// TwinCAT 3 PLC project Library
// Title: LCLS Sample Delivery
// Company: SLAC - LCLS
// ProjectVersion: 0.0.0
// ProgramVersion: 3.1.4023.0
// libraries:
//   LCLS Vacuum, * (SLAC - LCLS)
//   PMPS, * (SLAC - LCLS)
//   Tc2_EtherCAT, * (Beckhoff Automation GmbH)
//   Tc2_MC2, * (Beckhoff Automation GmbH)
//   Tc2_ModbusSrv, * (Beckhoff Automation GmbH)
//   Tc2_SerialCom, * (Beckhoff Automation GmbH)
//   Tc2_Standard, * (Beckhoff Automation GmbH)
//   Tc2_SUPS, * (Beckhoff Automation GmbH)
//   Tc2_System, * (Beckhoff Automation GmbH)
//   Tc2_Utilities, * (Beckhoff Automation GmbH)
//   Tc3_Module, * (Beckhoff Automation GmbH)
//   TcUnit, * (www.tcunit.org)
//   LCLS General,2.12.0,SLAC
// project tree:
//   DUTs/ALI/ E_AxisMoveMode.TcDUT (not stored), E_CTRL_MODE.TcDUT (not stored), E_PropValveFBState.TcDUT (not stored), HMI_PropValveCtrlState.TcDUT (not stored), ST_ALI.TcDUT (not stored), ST_ManipAxis.TcDUT (not stored), ST_PIDParams.TcDUT (not stored), ST_PressureController.TcDUT (not stored), ST_PropValveMKS253.TcDUT (not stored)
//   DUTs/Bronkhorst/ E_BHElFlowUnit.TcDUT (not stored), ST_BhElFlow.TcDUT (not stored)
//   DUTs/ E_AxisMotionState.TcDUT (not stored), ST_ManifoldValve.TcDUT (not stored), ST_Proportionair.TcDUT (not stored), ST_RegDeadbandControls.TcDUT (not stored), ST_Regulator.TcDUT (not stored), ST_SelectorM3.TcDUT (not stored), ST_Shaker.TcDUT (not stored), ST_ShakerControls.TcDUT (not stored), ST_Strings.TcDUT (not stored)
//   DUTs/General/ E_CTRL_MODE_1.TcDUT (not stored)
//   DUTs/IO_Structs/ ST_ALIIO.TcDUT (not stored), ST_M3DeviceBaseIO.TcDUT (not stored), ST_SerialComm.TcDUT (not stored)
//   DUTs/RCC/ E_RCC_PUMP_SM_STATES.TcDUT, E_RCC_STATES.TcDUT (not stored), ST_RCC.TcDUT
//   DUTs/Sensirion/ E_SensirionFMMode.TcTLEO (not stored), ST_SensirionFM.TcDUT (not stored), ST_SensirionFMControl.TcDUT (not stored), ST_SensirionFMStatus.TcDUT (not stored)
//   DUTs/TEC/ ST_TECControl.TcDUT (not stored), ST_TECStatus.TcDUT (not stored)
//   DUTs/Vici/EPS/ E_VICI_PORT_EPS.TcDUT, E_VICI_EPS_PORT_STATUS.TcDUT
//   DUTs/Vici/ ST_12ViciValveSampleNames.TcDUT, ST_4PViciValveSampleNames.TcDUT, ST_ViciControl.TcDUT (not stored), ST_ViciStatus.TcDUT (not stored)
//   GVLs/ GVL_SAMPLE.TcGVL (not stored)
//   / PlcTask.TcTTO (not stored)
//   POUs/ALI/ FB_ALI.TcPOU (not stored), FB_ManipAxis.TcPOU (not stored), FB_PID_EXT.TcPOU (not stored), FB_PropValve.TcPOU (not stored), F_AxisRef_To_MSTA.TcPOU (not stored), MC_SmoothMover.TcPOU (not stored)
//   POUs/Bronkhorst/ FB_BronkhorstMFM.TcPOU (not stored)
//   POUs/DigitalOutput/ FB_SolenoidPair.TcPOU (not stored)
//   POUs/ EXAMPLE_DEPLOYMENT.TcPOU (not stored), PRG_TEST.TcPOU
//   POUs/GasManifold/ FB_GasManifold.TcPOU (not stored), FB_ManiValve.TcPOU (not stored)
//   POUs/Helpers/ FB_EcatDiag.TcPOU (not stored), FB_SelectorSync.TcPOU (not stored), FB_SerialCommWrapper.TcPOU (not stored), FB_ShiftByteArray.TcPOU (not stored)
//   POUs/PCM/ FB_MPV1.TcPOU, FB_PCM_AIO.TcPOU, FB_PressureControlModule.TcPOU (not stored)
//   POUs/RCC/ FB_RCC.TcPOU (not stored), FB_RCC_PUMP.TcPOU, FB_RCC_SM.TcPOU (not stored), FB_VRC_NC_OPNLS.TcPOU (not stored)
//   POUs/Regulators/ FB_ProportionairRegulator.TcPOU (not stored), FB_Regulator.TcPOU (not stored), F_rPressure.TcPOU (not stored)
//   POUs/Selectors/ FB_SelectorM3.TcPOU (not stored)
//   POUs/Sensirion/ FB_SenserionFlowMeter.TcPOU (not stored), FB_SensirionDriver.TcPOU (not stored), FB_SensirionTransaction.TcPOU (not stored), fSHDLCChecksum.TcPOU (not stored)
//   POUs/TEC/ FB_TECDriver.TcPOU (not stored), FB_TECTransaction.TcPOU (not stored)
//   POUs/Tests/ FB_RCC_TEST.TcPOU (not stored), FB_VICI_EPS_TEST.TcPOU
//   POUs/VICI/EPS/ FB_12PVICI_EPS.TcPOU, FB_4PVICI_EPS.TcPOU, FB_ViciValveEPS.TcPOU, FB_VICI_EPS_LOGIC.TcPOU
//   POUs/VICI/ FB_12PortVici.TcPOU, FB_4PortViciValve.TcPOU (not stored), FB_ViciDriver.TcPOU (not stored), FB_ViciTransaction.TcPOU (not stored), FB_ViciValve.TcPOU (not stored)
// real-time tasks:
//   TASK PlcTask: cycle T#10ms, priority 20, ADS port 350

// ---- DUTs/RCC/E_RCC_PUMP_SM_STATES.TcDUT
{attribute 'qualified_only'}
{attribute 'strict'}
TYPE E_RCC_PUMP_SM_STATES :
(
    IDLE := 0,
    PRESSURE := 1,
    VACUUM := 2,
    VENT := 3
);
END_TYPE

// ---- DUTs/RCC/ST_RCC.TcDUT
TYPE ST_RCC :
STRUCT
    {attribute 'pytmc' :='
        pv: Tinterval
        io: io
        autosave_pass0: VAL DESC
    '} // Time before cycle starts
    TInterval : REAL := 10;
    {attribute 'pytmc' :='
        pv: T1
        io: io
        autosave_pass0: VAL DESC
    '}
    T1 : REAL := 20;
    {attribute 'pytmc' :='
        pv: T2
        io: io
        autosave_pass0: VAL DESC
    '}
    T2 : REAL := 10;
    {attribute 'pytmc' :='
        pv: T3
        io: io
        autosave_pass0: VAL DESC
    '}
    T3 : REAL := 5;
    {attribute 'pytmc' :='
        pv: T4
        io: io
        autosave_pass0: VAL DESC
    '}
    T4 : REAL := 10;
    {attribute 'pytmc' :=' pv: RUNCLEAN'}
    bRunClean : BOOL := TRUE;

    {attribute 'pytmc' :=' pv: CLEAR_ERROR'}
    bClearError : BOOL := FALSE;
    {attribute 'pytmc' :=' pv: ERROR'}
    bError : BOOL := FALSE;
    {attribute 'pytmc' :=' pv: STOP_CYCLE'}
    bStop : BOOL := FALSE;

    {attribute 'pytmc' :=' pv: START_CYCLE'}
    bStartCycle : BOOL  := FALSE;

    {attribute 'pytmc' :='
        pv: ILK_Setpoint
        autosave_pass0: VAL DESC
     '}
    RCC_GCP_01_INTERLOCK_SETPOINT : REAL := 10;
    {attribute 'pytmc' :=' pv: OverrideMode '}
    xSystemOverrideMode_RCC : BOOL := FALSE;

    eCurrentState : INT := E_RCC_STATES.IDLE;

    {attribute 'pytmc' :='
        pv: RCC_RUNNING
        io: o
    '}
    bRunning : BOOL := FALSE;
    {attribute 'pytmc' :='
        pv: RCC_TIMER
        io: o
    '}
    tTimerReadBack : STRING := '';
    {attribute 'pytmc' :=' pv: sLogMessage '}
    sLogMessage : T_MaxString := '';

    RCC_VRC_01_OPEN_OK : BOOL;
    RCC_VRC_02_OPEN_OK : BOOL;
    RCC_VRC_03_OPEN_OK : BOOL;
    RCC_VRC_04_OPEN_OK : BOOL;

END_STRUCT
END_TYPE

// ---- DUTs/Vici/EPS/E_VICI_PORT_EPS.TcDUT
TYPE E_VICI_PORT_EPS :
STRUCT
    {attribute 'pytmc' := 'pv: stEPS'}
    stEPS : DUT_EPS;
    {attribute 'pytmc' := 'pv: ePortStatus'}
    ePortStatus : E_VICI_EPS_PORT_STATUS;
END_STRUCT
END_TYPE

// ---- DUTs/Vici/EPS/E_VICI_EPS_PORT_STATUS.TcDUT
{attribute 'qualified_only'}
{attribute 'strict'}
TYPE E_VICI_EPS_PORT_STATUS :
(
    ACTIVE := 0,
    UNLOCKED := 1,
    LOCKED := 2
);
END_TYPE

// ---- DUTs/Vici/ST_12ViciValveSampleNames.TcDUT
TYPE ST_12ViciValveSampleNames :
STRUCT
    {attribute 'pytmc' := '
        pv: 01
        io: io
        autosave_pass0: VAL DESC
     '}
     s1 : STRING;
     {attribute 'pytmc' := '
        pv: 02
        io: io
        autosave_pass0: VAL DESC
     '}
     s2 : STRING;
     {attribute 'pytmc' := '
        pv: 03
        io: io
        autosave_pass0: VAL DESC
     '}
     s3 : STRING;
     {attribute 'pytmc' := '
        pv: 04
        io: io
        autosave_pass0: VAL DESC
     '}
     s4 : STRING;
           {attribute 'pytmc' := '
        pv: 05
        io: io
        autosave_pass0: VAL DESC
     '}
     s5 : STRING;
     {attribute 'pytmc' := '
        pv: 06
        io: io
        autosave_pass0: VAL DESC
     '}
     s6 : STRING;
     {attribute 'pytmc' := '
        pv: 07
        io: io
        autosave_pass0: VAL DESC
     '}
     s7 : STRING;
     {attribute 'pytmc' := '
        pv: 08
        io: io
        autosave_pass0: VAL DESC
     '}
     s8 : STRING;
           {attribute 'pytmc' := '
        pv: 09
        io: io
        autosave_pass0: VAL DESC
     '}
     s9 : STRING;
     {attribute 'pytmc' := '
        pv: 10
        io: io
        autosave_pass0: VAL DESC
     '}
     s10 : STRING;
     {attribute 'pytmc' := '
        pv: 11
        io: io
        autosave_pass0: VAL DESC
     '}
     s11 : STRING;
     {attribute 'pytmc' := '
        pv: 12
        io: io
        autosave_pass0: VAL DESC
     '}
     s12 : STRING;
END_STRUCT
END_TYPE

// ---- DUTs/Vici/ST_4PViciValveSampleNames.TcDUT
TYPE ST_4PViciValveSampleNames :
STRUCT
      {attribute 'pytmc' := '
        pv: 01
        io: io
        autosave_pass0: VAL DESC
     '}
     s1 : STRING;
     {attribute 'pytmc' := '
        pv: 02
        io: io
        autosave_pass0: VAL DESC
     '}
     s2 : STRING;
     {attribute 'pytmc' := '
        pv: 03
        io: io
        autosave_pass0: VAL DESC
     '}
     s3 : STRING;
     {attribute 'pytmc' := '
        pv: 04
        io: io
        autosave_pass0: VAL DESC
     '}
     s4 : STRING;
END_STRUCT
END_TYPE

// ---- POUs/PCM/FB_MPV1.TcPOU
FUNCTION_BLOCK FB_MPV1
(* Pressure Control Module 0-10v control and readback signal *)
VAR_INPUT
END_VAR
VAR_OUTPUT
END_VAR
VAR
    {attribute 'pytmc' := '
        pv: PropAir:01
     '}
    stPropAir1 : ST_Proportionair;
    {attribute 'pytmc' := '
        pv: PropAir:02
     '}
    stPropAir2 : ST_Proportionair;

    PropAir1 : FB_PCM_AIO;
    PropAir2 : FB_PCM_AIO;
END_VAR

PropAir1(iq_stRegProp:=stPropAir1, iDEVICE_MAX_PRESSURE := 100);
PropAir1(iq_stRegProp:=stPropAir1, iDEVICE_MAX_PRESSURE := 100);

END_FUNCTION_BLOCK

// ---- POUs/PCM/FB_PCM_AIO.TcPOU
FUNCTION_BLOCK FB_PCM_AIO
(* FUNCTION BLOCK FOR PRESSURE CONTROL MODULES WIT ANALOG IO CONTROL WITH 0-10v SIGNAL *)
VAR_INPUT
    iDEVICE_MAX_PRESSURE : INT := 100; // (psi)
END_VAR
VAR_OUTPUT
END_VAR
VAR
    iTermBits :INT := 32767;
END_VAR
VAR_IN_OUT
    iq_stRegProp	:	ST_Proportionair;
END_VAR

iq_stRegProp.iPressure := REAL_TO_INT(iDEVICE_MAX_PRESSURE * (MAX(0,INT_TO_REAL(iq_stRegProp.i_iPressRB)) / iTermBits));
iq_stRegProp.iSetpoint := LIMIT(iq_stRegProp.iLoLimit, iq_stRegProp.iSetpoint, iq_stRegProp.iHiLimit);
iq_stRegProp.q_iPressCt := REAL_TO_INT( (INT_TO_REAL(iq_stRegProp.iSetpoint)/iDEVICE_MAX_PRESSURE)*iTermBits);

END_FUNCTION_BLOCK

// ---- POUs/PRG_TEST.TcPOU
PROGRAM PRG_TEST
VAR
    fbRCC_TEST : FB_RCC_TEST;
    fbViciEPS_TEST : FB_VICI_EPS_TEST;
END_VAR

TcUnit.RUN();

END_PROGRAM

// ---- POUs/Tests/FB_VICI_EPS_TEST.TcPOU
FUNCTION_BLOCK FB_VICI_EPS_TEST EXTENDS FB_TestSuite
VAR_INPUT
END_VAR
VAR_OUTPUT
END_VAR
VAR

// TestEnableOverrideExpectOverrideToAutoRestAfterTimerExpires FBs
// These Fbs need to be defined outside of Test for Timers To Function Correcly.

    fbViciEPS : FB_VICI_EPS_LOGIC;
    aEPS : ARRAY[1..4] OF E_VICI_PORT_EPS;
    fbEPS : FB_EPS;
    bAllPortsLocked : BOOL;
    iReqNewPort : INT := 1;
    iNumPorts: INT := 4;
    bExternalSignal: BOOL;
    bOverride : BOOL := FALSE;
    fbTestTimer : TON;
    bTestInit : BOOL := TRUE;

	aEPS_4 : ARRAY[1..4] OF E_VICI_PORT_EPS;
	fb4PortViciEps : FB_4PVICI_EPS;
	aEPS_12 : ARRAY[1..12] OF E_VICI_PORT_EPS;
	fb12PortViciEps : FB_12PVICI_EPS;

END_VAR

TestRequestEpsNotOkPortExpectNoPortChange();
TestActivePortBecomesLockedExpectExternalSignalSetTrue();
TestAllPortsLockedExpectbAllPortsLockedToBeTrue();
TestEpsPortStatusChangeExpectPortStatusToChange();
TestLockedPortMovesWithOverrideExpectPortToMove();
TestEnableOverrideExpectOverrideToAutoRestAfterTimerExpires();


fb4PortViciEps(iAddress:=1, aPortEPS:=aEPS_4);
fb12PortViciEps(iAddress:=1, aPortEPS:=aEPS_12);

METHOD TestActivePortBecomesLockedExpectExternalSignalSetTrue :  REFERENCE TO FB_Test
VAR
    aEPS : ARRAY[1..4] OF E_VICI_PORT_EPS;
    fbViciEPS : FB_VICI_EPS_LOGIC;
    fbEPS : FB_EPS;

    bAllPortsLocked : BOOL;
    bExternalSignal : BOOL;
    iReqNewPort : INT;
    iNumPorts :INT := 4;
    bOverride : BOOL := FALSE;
END_VAR
TEST('TestActivePortBecomesLockedExpectExternalSignalSetTrue');

fbEPS(eps:=aEPS[1].stEPS);
fbEPS.setBit(0, TRUE);

fbEPS(eps:=aEPS[2].stEPS);
fbEPS.setBit(0, TRUE);

fbEPS(eps:=aEPS[3].stEPS);
fbEPS.setBit(0, TRUE);

fbEPS(eps:=aEPS[4].stEPS);
fbEPS.setBit(0, TRUE);

fbViciEPS(aPortEPS := aEPS,
    iReqPort := 1,
    iPrevPort := iReqNewPort,
    bOverride := bOverride,
    iNumPorts := iNumPorts,
    bExternalLockSignal => bExternalSignal,
    bAllPortsLocked => bAllPortsLocked,
    iNewPortPos => iReqNewPort);


AssertEquals_BOOL(
    Expected:= FALSE ,
    Actual:= bExternalSignal,
    Message:= 'bExternalSignal Should be FALSE'
);

fbEPS(eps:=aEPS[1].stEPS);
fbEPS.setBit(0, FALSE);

fbEPS(eps:=aEPS[2].stEPS);
fbEPS.setBit(0, TRUE);

fbEPS(eps:=aEPS[3].stEPS);
fbEPS.setBit(0, TRUE);

fbEPS(eps:=aEPS[4].stEPS);
fbEPS.setBit(0, TRUE);


fbViciEPS(aPortEPS := aEPS,
    iReqPort := 1,
    iPrevPort := iReqNewPort,
    bOverride := bOverride,
    iNumPorts := iNumPorts,
    bExternalLockSignal => bExternalSignal,
    bAllPortsLocked => bAllPortsLocked,
    iNewPortPos => iReqNewPort);


AssertEquals_BOOL(
    Expected:= TRUE ,
    Actual:= bExternalSignal,
    Message:= 'bExternalSignal Should be TRUE'
);

// CHECK OVERRIDE
bOverride := TRUE;

fbViciEPS(aPortEPS := aEPS,
    iReqPort := 1,
    iPrevPort := iReqNewPort,
    bOverride := bOverride,
    iNumPorts := iNumPorts,
    bExternalLockSignal => bExternalSignal,
    bAllPortsLocked => bAllPortsLocked,
    iNewPortPos => iReqNewPort);


AssertEquals_BOOL(
    Expected:= FALSE ,
    Actual:= bExternalSignal,
    Message:= 'bExternalSignal Should be FALSE'
);

TEST_FINISHED();
END_METHOD

METHOD TestAllPortsLockedExpectbAllPortsLockedToBeTrue :  REFERENCE TO FB_Test
VAR_INPUT
END_VAR
VAR
    fbViciEPS : FB_VICI_EPS_LOGIC;
    aEPS : ARRAY[1..4] OF E_VICI_PORT_EPS;

    fbEPS : FB_EPS;

    bAllPortsLocked : BOOL;
    iReqNewPort : INT;
    iNumPorts: INT := 4;
    bExternalSignal: BOOL;
    bOverride : BOOL := FALSE;
END_VAR
TEST('TestAllPortsLockedExpectbAllPortsLockedToBeTrue');
fbEPS(eps:=aEPS[1].stEPS);
fbEPS.setBit(0, TRUE);

fbEPS(eps:=aEPS[2].stEPS);
fbEPS.setBit(0, TRUE);

fbEPS(eps:=aEPS[3].stEPS);
fbEPS.setBit(0, TRUE);

fbEPS(eps:=aEPS[4].stEPS);
fbEPS.setBit(0, TRUE);

fbViciEPS(aPortEPS := aEPS,
    iReqPort := 1,
    iPrevPort := iReqNewPort,
    bOverride := bOverride,
    iNumPorts := iNumPorts,
    bExternalLockSignal => bExternalSignal,
    bAllPortsLocked => bAllPortsLocked,
    iNewPortPos => iReqNewPort);

AssertEquals_BOOL(
    Expected:= FALSE ,
    Actual:= bAllPortsLocked,
    Message:= 'ALL PORTS ARE LOCKED'
);

fbEPS(eps:=aEPS[1].stEPS);
fbEPS.setBit(0, FALSE);

fbEPS(eps:=aEPS[2].stEPS);
fbEPS.setBit(0, FALSE);

fbEPS(eps:=aEPS[3].stEPS);
fbEPS.setBit(0, FALSE);

fbEPS(eps:=aEPS[4].stEPS);
fbEPS.setBit(0, FALSE);

fbViciEPS(aPortEPS := aEPS,
    iReqPort := 1,
    iPrevPort := iReqNewPort,
    bOverride := bOverride,
    iNumPorts := iNumPorts,
    bExternalLockSignal => bExternalSignal,
    bAllPortsLocked => bAllPortsLocked,
    iNewPortPos => iReqNewPort);

AssertEquals_BOOL(
    Expected:= TRUE ,
    Actual:= bAllPortsLocked,
    Message:= 'ALL PORTS ARE NOT LOCKED'
);

TEST_FINISHED();
END_METHOD

METHOD TestEnableOverrideExpectOverrideToAutoRestAfterTimerExpires : REFERENCE TO FB_TEST
VAR_INPUT
END_VAR
TEST('TestEnableOverrideExpectOverrideToAutoRestAfterTimerExpires');

IF bTestInit THEN
    fbEPS(eps:=aEPS[1].stEPS);
    fbEPS.setBit(0, FALSE);

    fbEPS(eps:=aEPS[2].stEPS);
    fbEPS.setBit(0, FALSE);

    fbEPS(eps:=aEPS[3].stEPS);
    fbEPS.setBit(0, FALSE);

    fbEPS(eps:=aEPS[4].stEPS);
    fbEPS.setBit(0, TRUE);

    fbViciEPS.M_SET_OVERRIDE_RESET_TIME(tNewTime:=T#100ms);
    fbTestTimer.PT := T#500ms;
    fbTestTimer.IN := TRUE;

    // Enable Override
    bOverride := TRUE;

    // Move To Locked Port
    iReqNewPort := 1;

    fbViciEPS(aPortEPS := aEPS,
    iReqPort := iReqNewPort,
    iPrevPort := iReqNewPort,
    bOverride := bOverride,
    iNumPorts := iNumPorts,
    bExternalLockSignal => bExternalSignal,
    bAllPortsLocked => bAllPortsLocked,
    iNewPortPos => iReqNewPort);

    AssertEquals_INT(
    Expected:= E_VICI_EPS_PORT_STATUS.ACTIVE ,
    Actual:= aEPS[1].ePortStatus,
    Message:= 'PORT 1: NOT ACTIVE'
    );

    bTestInit := FALSE;

END_IF

fbViciEPS(aPortEPS := aEPS,
    iReqPort := iReqNewPort,
    iPrevPort := iReqNewPort,
    bOverride := bOverride,
    iNumPorts := iNumPorts,
    bExternalLockSignal => bExternalSignal,
    bAllPortsLocked => bAllPortsLocked,
    iNewPortPos => iReqNewPort);

IF  NOT bOverride OR fbTestTimer.Q THEN

    // Test if bOverride Reset.
    AssertEquals_BOOL(
    Expected:= FALSE ,
    Actual:= bOverride,
    Message:= 'bOverride was Not Reset');
	
	AssertEquals_BOOL(
    Expected:= FALSE ,
    Actual:= fbTestTimer.Q,
    Message:= 'TIMEOUT REACHED.');

    // TRY Blocked Move after override reset.
    iReqNewPort := 1;

    fbViciEPS(aPortEPS := aEPS,
    iReqPort := iReqNewPort,
    iPrevPort := iReqNewPort,
    bOverride := bOverride,
    iNumPorts := iNumPorts,
    bExternalLockSignal => bExternalSignal,
    bAllPortsLocked => bAllPortsLocked,
    iNewPortPos => iReqNewPort);

    AssertEquals_INT(
    Expected:= E_VICI_EPS_PORT_STATUS.LOCKED ,
    Actual:= aEPS[1].ePortStatus,
    Message:= 'PORT 1: IS ACTIVE'
    );

    TEST_FINISHED();
END_IF
END_METHOD

METHOD TestEpsPortStatusChangeExpectPortStatusToChange :  REFERENCE TO FB_Test
VAR_INPUT
END_VAR
VAR
    fbViciEPS : FB_VICI_EPS_LOGIC;
    aEPS : ARRAY[1..4] OF E_VICI_PORT_EPS;

    fbEPS : FB_EPS;

    bAllPortsLocked : BOOL;
    iReqNewPort : INT := 1;
    iNumPorts: INT := 4;
    bExternalSignal: BOOL;
    bOverride : BOOL := FALSE;
END_VAR
TEST('TestEpsPortStatusChangeExpectPortStatusToChange');
fbEPS(eps:=aEPS[1].stEPS);
fbEPS.setBit(0, TRUE);

fbEPS(eps:=aEPS[2].stEPS);
fbEPS.setBit(0, TRUE);

fbEPS(eps:=aEPS[3].stEPS);
fbEPS.setBit(0, TRUE);

fbEPS(eps:=aEPS[4].stEPS);
fbEPS.setBit(0, TRUE);

// MAKE PORT 1 ACTIVE
fbViciEPS(aPortEPS := aEPS,
    iReqPort := 1,
    iPrevPort := iReqNewPort,
    bOverride := bOverride,
    iNumPorts := iNumPorts,
    bExternalLockSignal => bExternalSignal,
    bAllPortsLocked => bAllPortsLocked,
    iNewPortPos => iReqNewPort);

AssertEquals_INT(
    Expected:= E_VICI_EPS_PORT_STATUS.ACTIVE ,
    Actual:= aEPS[1].ePortStatus,
    Message:= 'PORT 1: NOT ACTIVE'
);

// MAKE PORT 1 UNLOCKED

fbViciEPS(aPortEPS := aEPS,
    iReqPort := 2,
    iPrevPort := iReqNewPort,
    bOverride := bOverride,
    iNumPorts := iNumPorts,
    bExternalLockSignal => bExternalSignal,
    bAllPortsLocked => bAllPortsLocked,
    iNewPortPos => iReqNewPort);

AssertEquals_INT(
    Expected:= E_VICI_EPS_PORT_STATUS.UNLOCKED ,
    Actual:= aEPS[1].ePortStatus,
    Message:= 'PORT 1: NOT IN UNLOCKED STATE'
);

// MAKE PORT 1 LOCKED
fbEPS(eps:=aEPS[1].stEPS);
fbEPS.setBit(0, FALSE);

fbViciEPS(aPortEPS := aEPS,
    iReqPort := 2,
    iPrevPort := iReqNewPort,
    bOverride := bOverride,
    iNumPorts := iNumPorts,
    bExternalLockSignal => bExternalSignal,
    bAllPortsLocked => bAllPortsLocked,
    iNewPortPos => iReqNewPort);

AssertEquals_INT(
    Expected:= E_VICI_EPS_PORT_STATUS.LOCKED ,
    Actual:= aEPS[1].ePortStatus,
    Message:= 'PORT 1: NOT IN LOCKED STATE'
);

TEST_FINISHED();
END_METHOD

METHOD TestLockedPortMovesWithOverrideExpectPortToMove :  REFERENCE TO FB_Test
VAR_INPUT
END_VAR
VAR
    fbViciEPS : FB_VICI_EPS_LOGIC;
    aEPS : ARRAY[1..4] OF E_VICI_PORT_EPS;

    fbEPS : FB_EPS;
    bAllPortsLocked : BOOL;
    iReqNewPort : INT;
    iNumPorts : INT := 4;
    bExternalSignal: BOOL;
    bOverride : BOOL := FALSE;

    fbTestTimer : TON;
    iCount : INT := 0;
END_VAR
TEST('TestLockedPortMovesWithOverrideExpectPortToMove');
fbEPS(eps:=aEPS[1].stEPS);
fbEPS.setBit(0, TRUE);

fbEPS(eps:=aEPS[2].stEPS);
fbEPS.setBit(0, TRUE);

fbEPS(eps:=aEPS[3].stEPS);
fbEPS.setBit(0, FALSE);

fbEPS(eps:=aEPS[4].stEPS);
fbEPS.setBit(0, TRUE);

// REQUEST PORT 1
fbViciEPS(aPortEPS := aEPS,
    iReqPort := 1,
    iPrevPort := iReqNewPort,
    bOverride := bOverride,
    iNumPorts := iNumPorts,
    bExternalLockSignal => bExternalSignal,
    bAllPortsLocked => bAllPortsLocked,
    iNewPortPos => iReqNewPort);

AssertEquals_INT(Expected:= 1 ,
    Actual:= iReqNewPort,
    Message:= 'VICI EPS DID NOT MOVE TO ALLOWED PORT');

// REQUEST PORT 3 w/ Override

bOverride := TRUE;

fbViciEPS(aPortEPS := aEPS,
    iReqPort := 3,
    iPrevPort := iReqNewPort,
    bOverride := bOverride,
    iNumPorts := iNumPorts,
    bExternalLockSignal => bExternalSignal,
    bAllPortsLocked => bAllPortsLocked,
    iNewPortPos => iReqNewPort);

AssertEquals_INT(Expected:= 3 ,
    Actual:= iReqNewPort,
    Message:= 'VICI EPS OVERRIDE FAILED');

TEST_FINISHED();
END_METHOD

METHOD TestRequestEpsNotOkPortExpectNoPortChange :  REFERENCE TO FB_Test
VAR_INPUT
END_VAR
VAR
    fbViciEPS : FB_VICI_EPS_LOGIC;
    aEPS : ARRAY[1..4] OF E_VICI_PORT_EPS;
    fbEPS : FB_EPS;
    bAllPortsLocked : BOOL;
    iReqNewPort : INT;
    iNumPorts : INT := 4;
    bExternalSignal : BOOL;
    bOverride : BOOL := FALSE;
END_VAR
TEST('TestRequestEpsNotOkPortExpectNoPortChange');

fbEPS(eps:=aEPS[1].stEPS);
fbEPS.setBit(0, TRUE);

fbEPS(eps:=aEPS[2].stEPS);
fbEPS.setBit(0, TRUE);

fbEPS(eps:=aEPS[3].stEPS);
fbEPS.setBit(0, FALSE);

fbEPS(eps:=aEPS[4].stEPS);
fbEPS.setBit(0, TRUE);

// REQUEST PORT 1
fbViciEPS(aPortEPS := aEPS,
    iReqPort := 1,
    iPrevPort := iReqNewPort,
    bOverride := bOverride,
    iNumPorts := iNumPorts,
    bExternalLockSignal => bExternalSignal,
    bAllPortsLocked => bAllPortsLocked,
    iNewPortPos => iReqNewPort);

AssertEquals_INT(Expected:= 1 ,
    Actual:= iReqNewPort,
    Message:= 'VICI EPS DID NOT MOVE TO ALLOWED PORT');

// REQUEST PORT 3
fbViciEPS(aPortEPS := aEPS,
    iReqPort := 3,
    iPrevPort := iReqNewPort,
    bOverride := bOverride,
    iNumPorts := iNumPorts,
    bExternalLockSignal => bExternalSignal,
    bAllPortsLocked => bAllPortsLocked,
    iNewPortPos => iReqNewPort);

AssertEquals_INT(Expected:= 1 ,
    Actual:= iReqNewPort,
    Message:= 'VICI EPS MOVED TO BLOCKED PORT');


TEST_FINISHED();
END_METHOD

END_FUNCTION_BLOCK

// ---- POUs/VICI/EPS/FB_VICI_EPS_LOGIC.TcPOU
FUNCTION_BLOCK FB_VICI_EPS_LOGIC
VAR_INPUT
    iReqPort : INT;
    iPrevPort : INT;
    iNumPorts : INT;
END_VAR
VAR_IN_OUT
    aPortEPS : ARRAY [*] OF E_VICI_PORT_EPS; // EPS for each port.
    bOverride : BOOL;
END_VAR
VAR_OUTPUT
    bAllPortsLocked : BOOL;
    bExternalLockSignal : BOOL; // Signals if previously active port becomes locked.
    iNewPortPos : INT;
    tEPS_TimerCountDown : STRING;
END_VAR
VAR
    fbTimer : TON;
    tEPS_OVRD_RESET_TIME : TIME := T#1m;
    fbEPS : FB_EPS;
    iIndex : INT := 1;
    iEPS_NOT_OK_COUNT : INT;

END_VAR

M_RESET_EPS_TIMER();

// Evaluate all EPS
FOR iIndex := 1 TO iNumPorts BY 1 DO

    fbEPS(eps := aPortEPS[iIndex].stEPS);

    IF aPortEPS[iIndex].stEPS.bEPS_OK THEN
        aPortEPS[iIndex].ePortStatus := E_VICI_EPS_PORT_STATUS.UNLOCKED;
    ELSE
        aPortEPS[iIndex].ePortStatus := E_VICI_EPS_PORT_STATUS.LOCKED;
        iEPS_NOT_OK_COUNT := iEPS_NOT_OK_COUNT + 1;
    END_IF

END_FOR

iNewPortPos := iPrevPort;
IF aPortEPS[iReqPort].stEPS.bEPS_OK OR bOverride THEN
    iNewPortPos := iReqPort;
    aPortEPS[iReqPort].ePortStatus := E_VICI_EPS_PORT_STATUS.ACTIVE;
END_IF

IF (iReqPort = iPrevPort) AND (aPortEPS[iPrevPort].ePortStatus = E_VICI_EPS_PORT_STATUS.LOCKED) AND NOT bOverride THEN
    bExternalLockSignal := TRUE;
ELSIF  (iReqPort = iPrevPort) AND (aPortEPS[iPrevPort].ePortStatus <> E_VICI_EPS_PORT_STATUS.LOCKED) OR bOverride THEN
    bExternalLockSignal := FALSE;
END_IF

IF iEPS_NOT_OK_COUNT = iNumPorts AND NOT bOverride THEN
    bAllPortsLocked := TRUE;
ELSE
    bAllPortsLocked := FALSE;
END_IF

iIndex := 1;
iEPS_NOT_OK_COUNT := 0;

METHOD M_RESET_EPS_TIMER : BOOL
VAR_INPUT
END_VAR
fbTimer(IN := bOverride, PT:= tEPS_OVRD_RESET_TIME);

IF bOverride THEN
    tEPS_TimerCountDown := TIME_TO_STRING(tEPS_OVRD_RESET_TIME - fbTimer.ET);
END_IF

IF fbTimer.Q THEN
    bOverride := FALSE;
    tEPS_TimerCountDown := TIME_TO_STRING(T#0s);
END_IF
END_METHOD

METHOD M_SET_OVERRIDE_RESET_TIME : BOOL
VAR_INPUT
    tNewTime : TIME;
END_VAR
tEPS_OVRD_RESET_TIME := tNewTime;
END_METHOD

END_FUNCTION_BLOCK

// ---- POUs/VICI/EPS/FB_4PVICI_EPS.TcPOU
FUNCTION_BLOCK FB_4PVICI_EPS
VAR_INPUT
    iAddress : INT;
END_VAR
VAR_OUTPUT
    bAllPortsLocked : BOOL;
    bExternalLock : BOOL;
END_VAR
VAR_IN_OUT
    aPortEPS : ARRAY [*] OF E_VICI_PORT_EPS; // EPS for each port.
END_VAR
VAR

    {attribute 'pytmc' := '
        pv: ''
        io: io
    '}
    fbNporValveEPS : FB_ViciValveEPS;
    iNumPorts : INT := 4;

    {attribute 'pytmc' := '
        pv: SampleNames
        io: io
     '}
    stSampleNames : ST_4PViciValveSampleNames;

END_VAR

fbNporValveEPS(iAddress := iAddress,
    iNumOfPorts := iNumPorts,
    aPortEPS := aPortEPS,
    bAllPortsLocked => bAllPortsLocked,
    bExternalLock => bExternalLock);

END_FUNCTION_BLOCK

// ---- POUs/VICI/EPS/FB_ViciValveEPS.TcPOU
FUNCTION_BLOCK FB_ViciValveEPS
VAR_INPUT
    iAddress : INT;
    iNumOfPorts : INT;
END_VAR
VAR_IN_OUT
    aPortEPS : ARRAY [*] OF E_VICI_PORT_EPS; // EPS for each port.
END_VAR
VAR_OUTPUT
    bAllPortsLocked : BOOL;
    bExternalLock : BOOL;
END_VAR
VAR
    {attribute 'pytmc' := '
        pv: iReqPos
        io: io
     '}
    iReqPos : INT;

    {attribute 'pytmc' := '
    pv: PORT
    io: o
    '}
    iNewPortPos : INT;
    {attribute 'pytmc' := '
    pv: EPS
    io: o
    '}
    fbViciEPS : FB_VICI_EPS_LOGIC;

    {attribute 'pytmc' := 'pv: OVRD_MODE'}
    bEPS_Override : BOOL := FALSE;

    {attribute 'pytmc' := 'pv: OVRD_COUNTDOWN'}
    tEPS_TimerCountDown : STRING := TIME_TO_STRING(T#0s);

    fbNporValve : FB_ViciValve;
END_VAR

iReqPos := LIMIT(1,iReqPos, iNumOfPorts); // KEEP EPS array index within bounds

fbViciEPS(aPortEPS := aPortEPS,
    iReqPort := iReqPos,
    iPrevPort := iNewPortPos,
    bOverride := bEPS_Override,
    iNumPorts := iNumOfPorts,
    bExternalLockSignal => bExternalLock,
    bAllPortsLocked => bAllPortsLocked,
    iNewPortPos => iNewPortPos,
    tEPS_TimerCountDown => tEPS_TimerCountDown);

iReqPos := iNewPortPos; // Update iReqPos PV  to be the safe port, otherwise when EPS is cleared the requested port would automatically change.

fbNporValve(iAddress := iAddress,
            iNumOfPorts := iNumOfPorts,
            iReqPos := iNewPortPos);

END_FUNCTION_BLOCK

// ---- POUs/VICI/EPS/FB_12PVICI_EPS.TcPOU
FUNCTION_BLOCK FB_12PVICI_EPS
VAR_INPUT
    iAddress : INT;
END_VAR
VAR_OUTPUT
    bAllPortsLocked : BOOL;
    bExternalLock : BOOL;
END_VAR
VAR_IN_OUT
    aPortEPS : ARRAY [*] OF E_VICI_PORT_EPS; // EPS for each port.
END_VAR
VAR
    {attribute 'pytmc' := '
        pv: ''
        io: io
    '}
    fbNporValveEPS : FB_ViciValveEPS;
    iNumPorts : INT := 12;

    {attribute 'pytmc' := '
        pv: SampleNames
        io: io
     '}
    stSampleNames : ST_12ViciValveSampleNames;

END_VAR

fbNporValveEPS(iAddress := iAddress,
    iNumOfPorts := iNumPorts,
    aPortEPS := aPortEPS,
    bAllPortsLocked => bAllPortsLocked,
    bExternalLock => bExternalLock);

END_FUNCTION_BLOCK

// ---- POUs/RCC/FB_RCC_PUMP.TcPOU
(*This is a funcitonal prototype for in AIR RCC PUMP / L.V. RCC / WIP NAME*)
FUNCTION_BLOCK FB_RCC_PUMP
VAR_IN_OUT
    stRCC_VRC_01 : ST_VRC;
    stRCC_VRC_02 : ST_VRC;
    stRCC_VRC_03 : ST_VRC;

    T1 : TIME;
    T2 : TIME;
    T3 : TIME;

    bStart 	: BOOL := FALSE;
    bStop	: BOOL := FALSE;

END_VAR
VAR_OUTPUT
END_VAR
VAR
    iState 	: INT := E_RCC_PUMP_SM_STATES.IDLE;
    tTimer1 : TON;
    tTime : TIME := T#0s;
END_VAR

tTimer1(IN:=TRUE, PT:= tTime);

IF bStop THEN
    bStop := FALSE;
    stRCC_VRC_01.pv_xOPN_SW := FALSE;
    stRCC_VRC_02.pv_xOPN_SW := FALSE;
    stRCC_VRC_03.pv_xOPN_SW := FALSE;
    iState := E_RCC_PUMP_SM_STATES.IDLE;
END_IF

CASE iState OF
    E_RCC_PUMP_SM_STATES.IDLE: // IDlE

    IF bStart THEN
        iState := E_RCC_PUMP_SM_STATES.PRESSURE;
        bStart := FALSE;
        tTime := T1;
        tTimer1(IN:=FALSE); // RESTART TIMER
    END_IF

    E_RCC_PUMP_SM_STATES.PRESSURE: // PRESSURE

    stRCC_VRC_01.pv_xOPN_SW := FALSE;
    stRCC_VRC_02.pv_xOPN_SW := FALSE;
    stRCC_VRC_03.pv_xOPN_SW := TRUE;

    IF tTimer1.Q THEN
        iState := E_RCC_PUMP_SM_STATES.VACUUM;
        tTime := T2;
        tTimer1(IN:=FALSE); // RESTART TIMER
    END_IF

    E_RCC_PUMP_SM_STATES.VACUUM: // VACUUM

    stRCC_VRC_01.pv_xOPN_SW := FALSE;
    stRCC_VRC_02.pv_xOPN_SW := TRUE;
    stRCC_VRC_03.pv_xOPN_SW := FALSE;

    IF tTimer1.Q THEN
        iState := E_RCC_PUMP_SM_STATES.VENT;
        tTime := T3;
        tTimer1(IN:=FALSE); // RESTART TIMER
    END_IF

    E_RCC_PUMP_SM_STATES.VENT: // VENT;

    stRCC_VRC_01.pv_xOPN_SW := TRUE;
    stRCC_VRC_02.pv_xOPN_SW := FALSE;
    stRCC_VRC_03.pv_xOPN_SW := FALSE;

    IF tTimer1.Q THEN
        iState := E_RCC_PUMP_SM_STATES.VENT;
    END_IF

END_CASE

END_FUNCTION_BLOCK

// ---- POUs/VICI/FB_12PortVici.TcPOU
FUNCTION_BLOCK FB_12PortVici
VAR_INPUT
    iAddress : INT;
END_VAR
VAR_OUTPUT
END_VAR
VAR
    fbNporValve : FB_ViciValve;
    iNumPorts : INT := 12;

    {attribute 'pytmc' := '
        pv: iReqPos
        io: io
     '}
    iReqPos : INT;
    {attribute 'pytmc' := '
        pv: SampleNames
        io: io
     '}
    stSampleNames : ST_12ViciValveSampleNames;
END_VAR

fbNporValve(iAddress := iAddress, iNumOfPorts := iNumPorts, iReqPos := iReqPos);

END_FUNCTION_BLOCK
